PROGRAM PRG_ExtruderSys_Alt
VAR
	fbExtrusionSystem: FB_ExtrusionSystemRev;
END_VAR

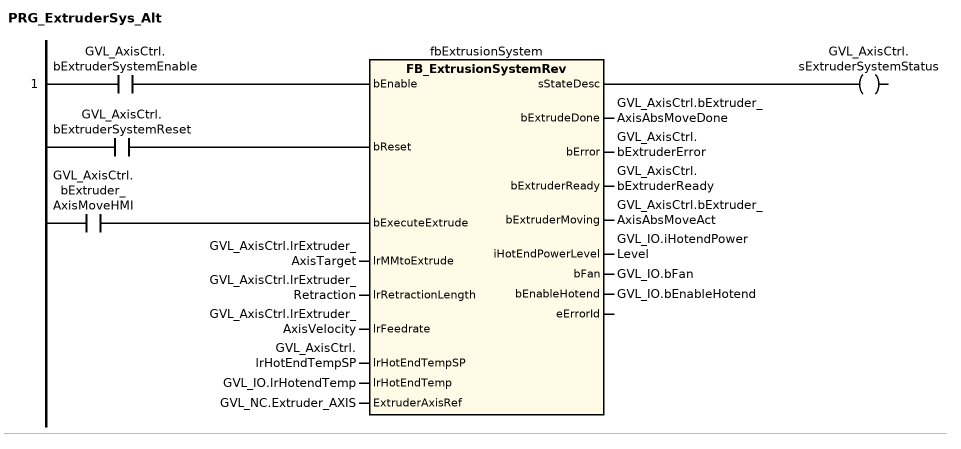
// NETWORK 1
fbExtrusionSystem(
    bEnable := GVL_AxisCtrl.bExtruderSystemEnable,
    bReset := GVL_AxisCtrl.bExtruderSystemReset,
    bExecuteExtrude := GVL_AxisCtrl.bExtruder_AxisMoveHMI,
    lrMMtoExtrude := GVL_AxisCtrl.lrExtruder_AxisTarget,
    lrRetractionLength := GVL_AxisCtrl.lrExtruder_Retraction,
    lrFeedrate := GVL_AxisCtrl.lrExtruder_AxisVelocity,
    lrHotEndTempSP := GVL_AxisCtrl.lrHotEndTempSP,
    lrHotEndTemp := GVL_IO.lrHotendTemp,
    ExtruderAxisRef := GVL_NC.Extruder_AXIS,
    bExtrudeDone => GVL_AxisCtrl.bExtruder_AxisAbsMoveDone,
    bError => GVL_AxisCtrl.bExtruderError,
    bExtruderReady => GVL_AxisCtrl.bExtruderReady,
    bExtruderMoving => GVL_AxisCtrl.bExtruder_AxisAbsMoveAct,
    iHotEndPowerLevel => GVL_IO.iHotendPowerLevel,
    bFan => GVL_IO.bFan,
    bEnableHotend => GVL_IO.bEnableHotend); // FB_ExtrusionSystemRev
GVL_AxisCtrl.sExtruderSystemStatus := fbExtrusionSystem.sStateDesc;

END_PROGRAM

(* stored: Version 1.1.0.1, ProductVersion 3.1.4024.2
   POU PRG_ExtruderSys_Alt: Id {b315064a-5d3a-40fb-bb21-0bb3a9d071d6}, SpecialFunc None *)
